FUNCTION_BLOCK Cylinder 
VAR_INPUT
END_VAR
VAR_OUTPUT
	bExtended : BOOL;
	bExtend : BOOL;
END_VAR
VAR
	fbExtendedSignal : BoolIn;
	fbExtend : BoolOut;
END_VAR

bExtended := fbExtendedSignal.getValue;
bExtend := fbExtend.getValue;

PROPERTY getExtend : BoolOut
GET
getExtend := fbExtend;
END_GET
END_PROPERTY

END_FUNCTION_BLOCK

(* stored: Version 1.1.0.1, ProductVersion 3.1.4024.0
   POU Cylinder: Id {4dff6417-8bf1-4724-a444-43bb6b5867e9}, SpecialFunc None
   Property getExtend: Id {551c2e8d-9793-498c-9e33-32fe5f29706c}
   Get Get: Id {70090b27-bd92-4955-9176-2f006b2ffbdc} *)
